// TIA Portal V16 export
// export: Created 2021-09-08T12:46:15.3662291Z, ExportSetting WithDefaults, DisplayName Totally Integrated Automation Portal, DisplayVersion V16 Update 3, DisplayName TIA Portal Version Control Interface, DisplayVersion V16 Update 2, DisplayName TIA Portal Openness, DisplayVersion V16 Update 3, DisplayName TIA Portal Teamcenter Gateway, DisplayVersion V16, DisplayName STEP 7 Professional, DisplayVersion V16 Update 3, DisplayName STEP 7 Safety, DisplayVersion V16, DisplayName WinCC Advanced, DisplayVersion V16 Update 3
DATA_BLOCK "AllPID_DB"   // DB11
VERSION : 0.1
// stored: AutoNumber true, DBAccessibleFromOPCUA true, InstanceOfName AllPID, InstanceOfType FB
"AllPID"
   // VAR
   //    P30x { S7_SetPoint := 'True'} : "PID_Pump2Pu1Fc";
   //    P120x { S7_SetPoint := 'True'} : "PID_Pump2Pu1Fc";
   //    P150x { S7_SetPoint := 'True'} : "PID_Pump2Pu1Fc";
   //    P901 { S7_SetPoint := 'True'} : "PID_Pump";
   //    P1301 { S7_SetPoint := 'True'} : "PID_Pump";
   // END_VAR
BEGIN
END_DATA_BLOCK
